{attribute 'GeneratedUsingTerminal: EL3413-0000-0016'}
{attribute addProperty BoxType "EL3413-0000-0016"}
{attribute addProperty Id "STATUSAT %I*STATUS_522E84CD1IndexAT %I*USINT1ChannelAT %I*USINT1ValueAT %I*DINT4"}
{attribute addProperty CRC "959271179"}
{attribute addProperty Size "7"}
TYPE PM_Inputs_Auxiliary_392D510B :
STRUCT
	{attribute addProperty Name "STATUS"}
	STATUS AT %I* : STATUS_522E84CD;
	{attribute addProperty Name "Index"}
	Index AT %I* : USINT;
	{attribute addProperty Name "Channel"}
	Channel AT %I* : USINT;
	{attribute addProperty Name "Value"}
	Value AT %I* : DINT;
END_STRUCT
END_TYPE

(* stored: Version 1.2.0.0, ProductVersion 3.1.4024.9
   DUT PM_Inputs_Auxiliary_392D510B: Id {3fd74fb7-2332-4c0f-9732-d0be355d05e7} *)
